PROGRAM PRG_HV_ILK
VAR
	HV_ILK_OK: bool := false;
END_VAR


//evaluate the HV ILK_OK bit
//HV_ILK_OK := GCC_40.IG.xAT_VAC;

hv1(i_xExtIlkOK := HV_ILK_OK);
hv2(i_xExtIlkOK := HV_ILK_OK);

END_PROGRAM

(* stored: Version 1.1.0.1, ProductVersion 3.1.4022.12
   POU PRG_HV_ILK: Id {b7f9d5cf-3c12-4ed0-bda8-0127f560a4d0}, SpecialFunc None *)
